FUNCTION_BLOCK CROSSCOMM_SENDER_209BB7FF9E1CBD715 (* Service Interface Function Block Type *)
  (* Standard: 61499-2 *)
  (* Version 0.0, 9/22/2017, bababen, nxtControl GmbH, template *)
  PACKAGE Main;
  (* Compiler Cpp nxtControl builtin 1.0 *)
  {SET_ATTRIBUTE(Runtime.FBType.ImplementingType, Runtime.System#DYNGEN_CROSSCOMM_SENDER)}
  {SET_ATTRIBUTE(Configuration.GenericFBType.InterfaceParams, Runtime.System#<InterfaceList> <EventInputs> <Event Name="LEXTEND" /> <Event Name="LRETRACT" /> </EventInputs> <InputVars /> </InterfaceList>)}
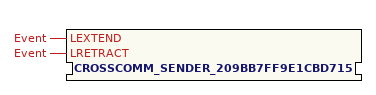
  EVENT_INPUT
    LEXTEND;
    LRETRACT;
  END_EVENT
  EC_STATES
    START;
  END_STATES
END_FUNCTION_BLOCK
